        ! Point 24: (200, 700) [rapid], axis_6=0
        CurrentX:=200;
        CurrentY:=700;
        pCurrent.trans:=[-1*CurrentX,CurrentY,SafeZ];
        pCurrent.rot:=OrientZYX(0,20,180);
        pCurrent.robconf:=[1,0,-2,0];
        TcpWorldX:=Bed1Wyong.uframe.trans.x+pCurrent.trans.x;
        CalcTrack:=TcpWorldX;
        IF CurrentY<1000 THEN CalcTrack:=CalcTrack+1500; ENDIF
        IF CurrentY<=1500 THEN
            IF (CalcTrack-TcpWorldX)<MinTrackSep THEN CalcTrack:=TcpWorldX+MinTrackSep; ENDIF
        ENDIF
        IF CalcTrack<TrackMin THEN CalcTrack:=TrackMin; ENDIF
        IF CalcTrack>TrackMax THEN CalcTrack:=TrackMax; ENDIF
        pCurrent.extax:=[CalcTrack,9E+09,9E+09,9E+09,9E+09,9E+09];
        MoveJ pCurrent,v500,z5,tVac\WObj:=Bed1Wyong;

        ! Point 25: (200, 700) [rapid], axis_6=180
        CurrentX:=200;
        CurrentY:=700;
        pCurrent.trans:=[-1*CurrentX,CurrentY,SafeZ];
        pCurrent.rot:=OrientZYX(180,20,180);
        pCurrent.robconf:=[1,0,0,0];
        TcpWorldX:=Bed1Wyong.uframe.trans.x+pCurrent.trans.x;
        CalcTrack:=TcpWorldX;
        IF CurrentY<1000 THEN CalcTrack:=CalcTrack+1500; ENDIF
        IF CurrentY<=1500 THEN
            IF (CalcTrack-TcpWorldX)<MinTrackSep THEN CalcTrack:=TcpWorldX+MinTrackSep; ENDIF
        ENDIF
        IF CalcTrack<TrackMin THEN CalcTrack:=TrackMin; ENDIF
        IF CalcTrack>TrackMax THEN CalcTrack:=TrackMax; ENDIF
        pCurrent.extax:=[CalcTrack,9E+09,9E+09,9E+09,9E+09,9E+09];
        MoveJ pCurrent,v500,z5,tVac\WObj:=Bed1Wyong;

        ! Descend to work height
        pCurrent.trans.z:=WorkZ;
        MoveL pCurrent,v100,z1000,tVac\WObj:=Bed1Wyong;

        ! Point 26: (200, 700) [work], axis_6=180
        CurrentX:=200;
        CurrentY:=700;
        pCurrent.trans:=[-1*CurrentX,CurrentY,WorkZ];
        pCurrent.rot:=OrientZYX(180,20,180);
        pCurrent.robconf:=[1,0,0,0];
        TcpWorldX:=Bed1Wyong.uframe.trans.x+pCurrent.trans.x;
        CalcTrack:=TcpWorldX;
        IF CurrentY<1000 THEN CalcTrack:=CalcTrack+1500; ENDIF
        IF CurrentY<=1500 THEN
            IF (CalcTrack-TcpWorldX)<MinTrackSep THEN CalcTrack:=TcpWorldX+MinTrackSep; ENDIF
        ENDIF
        IF CalcTrack<TrackMin THEN CalcTrack:=TrackMin; ENDIF
        IF CalcTrack>TrackMax THEN CalcTrack:=TrackMax; ENDIF
        pCurrent.extax:=[CalcTrack,9E+09,9E+09,9E+09,9E+09,9E+09];
        MoveL pCurrent,vTravel,z200,tVac\WObj:=Bed1Wyong;

        ! Point 27: (8050, 700) [work], axis_6=180
        CurrentX:=8050;
        CurrentY:=700;
        pCurrent.trans:=[-1*CurrentX,CurrentY,WorkZ];
        pCurrent.rot:=OrientZYX(180,20,180);
        pCurrent.robconf:=[1,0,0,0];
        TcpWorldX:=Bed1Wyong.uframe.trans.x+pCurrent.trans.x;
        CalcTrack:=TcpWorldX;
        IF CurrentY<1000 THEN CalcTrack:=CalcTrack+1500; ENDIF
        IF CurrentY<=1500 THEN
            IF (CalcTrack-TcpWorldX)<MinTrackSep THEN CalcTrack:=TcpWorldX+MinTrackSep; ENDIF
        ENDIF
        IF CalcTrack<TrackMin THEN CalcTrack:=TrackMin; ENDIF
        IF CalcTrack>TrackMax THEN CalcTrack:=TrackMax; ENDIF
        pCurrent.extax:=[CalcTrack,9E+09,9E+09,9E+09,9E+09,9E+09];
        MoveL pCurrent,vTravel,z200,tVac\WObj:=Bed1Wyong;

        ! Point 28: (8050, 500) [rapid], axis_6=180
        CurrentX:=8050;
        CurrentY:=500;
        pCurrent.trans:=[-1*CurrentX,CurrentY,SafeZ];
        pCurrent.rot:=OrientZYX(180,20,180);
        pCurrent.robconf:=[1,0,0,0];
        TcpWorldX:=Bed1Wyong.uframe.trans.x+pCurrent.trans.x;
        CalcTrack:=TcpWorldX;
        IF CurrentY<1000 THEN CalcTrack:=CalcTrack+1500; ENDIF
        IF CurrentY<=1500 THEN
            IF (CalcTrack-TcpWorldX)<MinTrackSep THEN CalcTrack:=TcpWorldX+MinTrackSep; ENDIF
        ENDIF
        IF CalcTrack<TrackMin THEN CalcTrack:=TrackMin; ENDIF
        IF CalcTrack>TrackMax THEN CalcTrack:=TrackMax; ENDIF
        pCurrent.extax:=[CalcTrack,9E+09,9E+09,9E+09,9E+09,9E+09];
        MoveJ pCurrent,v500,z5,tVac\WObj:=Bed1Wyong;

        ! Point 29: (8050, 500) [rapid], axis_6=0
        CurrentX:=8050;
        CurrentY:=500;
        pCurrent.trans:=[-1*CurrentX,CurrentY,SafeZ];
        pCurrent.rot:=OrientZYX(0,20,180);
        pCurrent.robconf:=[1,0,-2,0];
        TcpWorldX:=Bed1Wyong.uframe.trans.x+pCurrent.trans.x;
        CalcTrack:=TcpWorldX;
        IF CurrentY<1000 THEN CalcTrack:=CalcTrack+1500; ENDIF
        IF CurrentY<=1500 THEN
            IF (CalcTrack-TcpWorldX)<MinTrackSep THEN CalcTrack:=TcpWorldX+MinTrackSep; ENDIF
        ENDIF
        IF CalcTrack<TrackMin THEN CalcTrack:=TrackMin; ENDIF
        IF CalcTrack>TrackMax THEN CalcTrack:=TrackMax; ENDIF
        pCurrent.extax:=[CalcTrack,9E+09,9E+09,9E+09,9E+09,9E+09];
        MoveJ pCurrent,v500,z5,tVac\WObj:=Bed1Wyong;

        ! Descend to work height
        pCurrent.trans.z:=WorkZ;
        MoveL pCurrent,v100,z1000,tVac\WObj:=Bed1Wyong;

        ! Point 30: (8050, 500) [work], axis_6=0
        CurrentX:=8050;
        CurrentY:=500;
        pCurrent.trans:=[-1*CurrentX,CurrentY,WorkZ];
        pCurrent.rot:=OrientZYX(0,20,180);
        pCurrent.robconf:=[1,0,-2,0];
        TcpWorldX:=Bed1Wyong.uframe.trans.x+pCurrent.trans.x;
        CalcTrack:=TcpWorldX;
        IF CurrentY<1000 THEN CalcTrack:=CalcTrack+1500; ENDIF
        IF CurrentY<=1500 THEN
            IF (CalcTrack-TcpWorldX)<MinTrackSep THEN CalcTrack:=TcpWorldX+MinTrackSep; ENDIF
        ENDIF
        IF CalcTrack<TrackMin THEN CalcTrack:=TrackMin; ENDIF
        IF CalcTrack>TrackMax THEN CalcTrack:=TrackMax; ENDIF
        pCurrent.extax:=[CalcTrack,9E+09,9E+09,9E+09,9E+09,9E+09];
        MoveL pCurrent,vTravel,z200,tVac\WObj:=Bed1Wyong;

        ! Point 31: (200, 500) [work], axis_6=0
        CurrentX:=200;
        CurrentY:=500;
        pCurrent.trans:=[-1*CurrentX,CurrentY,WorkZ];
        pCurrent.rot:=OrientZYX(0,20,180);
        pCurrent.robconf:=[1,0,-2,0];
        TcpWorldX:=Bed1Wyong.uframe.trans.x+pCurrent.trans.x;
        CalcTrack:=TcpWorldX;
        IF CurrentY<1000 THEN CalcTrack:=CalcTrack+1500; ENDIF
        IF CurrentY<=1500 THEN
            IF (CalcTrack-TcpWorldX)<MinTrackSep THEN CalcTrack:=TcpWorldX+MinTrackSep; ENDIF
        ENDIF
        IF CalcTrack<TrackMin THEN CalcTrack:=TrackMin; ENDIF
        IF CalcTrack>TrackMax THEN CalcTrack:=TrackMax; ENDIF
        pCurrent.extax:=[CalcTrack,9E+09,9E+09,9E+09,9E+09,9E+09];
        MoveL pCurrent,vTravel,z200,tVac\WObj:=Bed1Wyong;

        ! Point 32: (200, 400) [rapid], axis_6=0
        CurrentX:=200;
        CurrentY:=400;
        pCurrent.trans:=[-1*CurrentX,CurrentY,SafeZ];
        pCurrent.rot:=OrientZYX(0,20,180);
        pCurrent.robconf:=[1,0,-2,0];
        TcpWorldX:=Bed1Wyong.uframe.trans.x+pCurrent.trans.x;
        CalcTrack:=TcpWorldX;
        IF CurrentY<1000 THEN CalcTrack:=CalcTrack+1500; ENDIF
        IF CurrentY<=1500 THEN
            IF (CalcTrack-TcpWorldX)<MinTrackSep THEN CalcTrack:=TcpWorldX+MinTrackSep; ENDIF
        ENDIF
        IF CalcTrack<TrackMin THEN CalcTrack:=TrackMin; ENDIF
        IF CalcTrack>TrackMax THEN CalcTrack:=TrackMax; ENDIF
        pCurrent.extax:=[CalcTrack,9E+09,9E+09,9E+09,9E+09,9E+09];
        MoveJ pCurrent,v500,z5,tVac\WObj:=Bed1Wyong;

        ! Point 33: (200, 400) [rapid], axis_6=180
        CurrentX:=200;
        CurrentY:=400;
        pCurrent.trans:=[-1*CurrentX,CurrentY,SafeZ];
        pCurrent.rot:=OrientZYX(180,20,180);
        pCurrent.robconf:=[1,0,0,0];
        TcpWorldX:=Bed1Wyong.uframe.trans.x+pCurrent.trans.x;
        CalcTrack:=TcpWorldX;
        IF CurrentY<1000 THEN CalcTrack:=CalcTrack+1500; ENDIF
        IF CurrentY<=1500 THEN
            IF (CalcTrack-TcpWorldX)<MinTrackSep THEN CalcTrack:=TcpWorldX+MinTrackSep; ENDIF
        ENDIF
        IF CalcTrack<TrackMin THEN CalcTrack:=TrackMin; ENDIF
        IF CalcTrack>TrackMax THEN CalcTrack:=TrackMax; ENDIF
        pCurrent.extax:=[CalcTrack,9E+09,9E+09,9E+09,9E+09,9E+09];
        MoveJ pCurrent,v500,z5,tVac\WObj:=Bed1Wyong;

        ! Descend to work height
        pCurrent.trans.z:=WorkZ;
        MoveL pCurrent,v100,z1000,tVac\WObj:=Bed1Wyong;

        ! Point 34: (200, 400) [work], axis_6=180
        CurrentX:=200;
        CurrentY:=400;
        pCurrent.trans:=[-1*CurrentX,CurrentY,WorkZ];
        pCurrent.rot:=OrientZYX(180,20,180);
        pCurrent.robconf:=[1,0,0,0];
        TcpWorldX:=Bed1Wyong.uframe.trans.x+pCurrent.trans.x;
        CalcTrack:=TcpWorldX;
        IF CurrentY<1000 THEN CalcTrack:=CalcTrack+1500; ENDIF
        IF CurrentY<=1500 THEN
            IF (CalcTrack-TcpWorldX)<MinTrackSep THEN CalcTrack:=TcpWorldX+MinTrackSep; ENDIF
        ENDIF
        IF CalcTrack<TrackMin THEN CalcTrack:=TrackMin; ENDIF
        IF CalcTrack>TrackMax THEN CalcTrack:=TrackMax; ENDIF
        pCurrent.extax:=[CalcTrack,9E+09,9E+09,9E+09,9E+09,9E+09];
        MoveL pCurrent,vTravel,z200,tVac\WObj:=Bed1Wyong;

        ! Point 35: (8050, 400) [work], axis_6=180
        CurrentX:=8050;
        CurrentY:=400;
        pCurrent.trans:=[-1*CurrentX,CurrentY,WorkZ];
        pCurrent.rot:=OrientZYX(180,20,180);
        pCurrent.robconf:=[1,0,0,0];
        TcpWorldX:=Bed1Wyong.uframe.trans.x+pCurrent.trans.x;
        CalcTrack:=TcpWorldX;
        IF CurrentY<1000 THEN CalcTrack:=CalcTrack+1500; ENDIF
        IF CurrentY<=1500 THEN
            IF (CalcTrack-TcpWorldX)<MinTrackSep THEN CalcTrack:=TcpWorldX+MinTrackSep; ENDIF
        ENDIF
        IF CalcTrack<TrackMin THEN CalcTrack:=TrackMin; ENDIF
        IF CalcTrack>TrackMax THEN CalcTrack:=TrackMax; ENDIF
        pCurrent.extax:=[CalcTrack,9E+09,9E+09,9E+09,9E+09,9E+09];
        MoveL pCurrent,vTravel,z200,tVac\WObj:=Bed1Wyong;


        ! Lift to safe height (before motor off for smooth blend)
        pCurrent.trans.z:=WorkZ+500;
        MoveL pCurrent,v200,z1000,tVac\WObj:=Bed1Wyong;
        Vac_off;

        ! Return tool and go home
        TPWrite "Py2Vac: Dropping off tool...";
        Vac_Dropoff;
        Home FALSE;

        TPWrite "========================================";
        TPWrite "Py2Vac: COMPLETE";
        TPWrite "========================================";

    ERROR
        Vac_off;
        TPWrite "Py2Vac ERROR: " \Num:=ERRNO;
        RAISE;
    ENDPROC

    PROC Py2Pan()
        ! Py2Pan - Generated by Onyx Tool Class
        ! Workzone: panel
        ! Area: (500,500) to (1900,1800)
        ! Z = 451mm
        ! Step: 300mm

        VAR robtarget pCurrent;
        VAR jointtarget CurrentJoints;
        VAR robtarget CurrentPos;
        VAR num WorkZ:=451;
        VAR num SafeZ:=651;
        VAR num CurrentX:=0;
        VAR num CurrentY:=0;
        VAR speeddata vTravel:=[100,500,5000,1000];
        VAR num TrackMin:=-300;
        VAR num TrackMax:=10050;
        VAR num CalcTrack:=0;
        VAR zonedata z1000:=[FALSE,1000,1500,1500,150,1500,150];
        VAR num PanForce:=0;
        VAR bool bFCActive:=FALSE;

        TPWrite "========================================";
        TPWrite "Py2Pan: Starting";
        TPWrite "========================================";
        TPWrite "Workzone: panel";
        TPWrite "WorkZ=" \Num:=WorkZ;

        ! Get helicopter tool (Pan attaches to it)
        UpdateToolNum;
        IF ToolNum<>2 THEN
            TPWrite "Py2Pan: Getting helicopter...";
            Home TRUE;
            Heli_Pickup;
        ELSE
            CurrentJoints:=CJointT();
            CurrentPos:=CalcRobT(CurrentJoints,tHeli\WObj:=wobj0);
            IF (CurrentPos.trans.x)>8000 AND CurrentPos.trans.z<400 THEN
                MoveL Offs(CurrentPos,0,0,(400-CurrentPos.trans.z)),v100,z5,tHeli;
            ENDIF
        ENDIF

        ! Set blade angle = 0 for pan
        HeliBlade_Angle 0;

        ! Start blade rotation
        TPWrite "Py2Pan: Starting blades at " \Num:=80;
        HeliBladeSpeed 80,"REV";
        TPWrite "Py2Pan: Blades motor on";
        WaitTime 5;

        ! ========================================
        ! Pattern Execution: 24 points
        ! ========================================

        ! Point 1: (500, 1800) [rapid]
        CurrentX:=500;
        CurrentY:=1800;
        pCurrent.trans:=[-1*CurrentX,CurrentY,SafeZ];
        pCurrent.rot:=OrientZYX(0,0,180);
        pCurrent.robconf:=[1,0,-2,0];
        CalcTrack:=Bed1Wyong.uframe.trans.x+pCurrent.trans.x;
        IF CurrentY<1000 THEN CalcTrack:=CalcTrack+1200; ENDIF
        IF CalcTrack<TrackMin THEN CalcTrack:=TrackMin; ENDIF
        IF CalcTrack>TrackMax THEN CalcTrack:=TrackMax; ENDIF
        pCurrent.extax:=[CalcTrack,9E+09,9E+09,9E+09,9E+09,9E+09];
        MoveJ pCurrent,v500,z5,tHeli\WObj:=Bed1Wyong;

        ! Descend to work height
        pCurrent.trans.z:=WorkZ;
        MoveL pCurrent,v100,z1000,tHeli\WObj:=Bed1Wyong;

        ! Point 2: (1900, 1800) [work]
        CurrentX:=1900;
        CurrentY:=1800;
        pCurrent.trans:=[-1*CurrentX,CurrentY,WorkZ];
        pCurrent.rot:=OrientZYX(0,0,180);
        pCurrent.robconf:=[1,0,-2,0];
        CalcTrack:=Bed1Wyong.uframe.trans.x+pCurrent.trans.x;
        IF CurrentY<1000 THEN CalcTrack:=CalcTrack+1200; ENDIF
        IF CalcTrack<TrackMin THEN CalcTrack:=TrackMin; ENDIF
        IF CalcTrack>TrackMax THEN CalcTrack:=TrackMax; ENDIF
        pCurrent.extax:=[CalcTrack,9E+09,9E+09,9E+09,9E+09,9E+09];
        MoveL pCurrent,vTravel,z200,tHeli\WObj:=Bed1Wyong;

        ! Point 3: (1900, 1500) [work]
        CurrentX:=1900;
        CurrentY:=1500;
        pCurrent.trans:=[-1*CurrentX,CurrentY,WorkZ];
        pCurrent.rot:=OrientZYX(0,0,180);
        pCurrent.robconf:=[1,0,-2,0];
        CalcTrack:=Bed1Wyong.uframe.trans.x+pCurrent.trans.x;
        IF CurrentY<1000 THEN CalcTrack:=CalcTrack+1200; ENDIF
        IF CalcTrack<TrackMin THEN CalcTrack:=TrackMin; ENDIF
        IF CalcTrack>TrackMax THEN CalcTrack:=TrackMax; ENDIF
        pCurrent.extax:=[CalcTrack,9E+09,9E+09,9E+09,9E+09,9E+09];
        MoveL pCurrent,vTravel,z200,tHeli\WObj:=Bed1Wyong;

        ! Point 4: (500, 1500) [work]
        CurrentX:=500;
        CurrentY:=1500;
        pCurrent.trans:=[-1*CurrentX,CurrentY,WorkZ];
        pCurrent.rot:=OrientZYX(0,0,180);
        pCurrent.robconf:=[1,0,-2,0];
        CalcTrack:=Bed1Wyong.uframe.trans.x+pCurrent.trans.x;
        IF CurrentY<1000 THEN CalcTrack:=CalcTrack+1200; ENDIF
        IF CalcTrack<TrackMin THEN CalcTrack:=TrackMin; ENDIF
        IF CalcTrack>TrackMax THEN CalcTrack:=TrackMax; ENDIF
        pCurrent.extax:=[CalcTrack,9E+09,9E+09,9E+09,9E+09,9E+09];
        MoveL pCurrent,vTravel,z200,tHeli\WObj:=Bed1Wyong;

        ! Point 5: (500, 1200) [work]
        CurrentX:=500;
        CurrentY:=1200;
        pCurrent.trans:=[-1*CurrentX,CurrentY,WorkZ];
        pCurrent.rot:=OrientZYX(0,0,180);
        pCurrent.robconf:=[1,0,-2,0];
        CalcTrack:=Bed1Wyong.uframe.trans.x+pCurrent.trans.x;
        IF CurrentY<1000 THEN CalcTrack:=CalcTrack+1200; ENDIF
        IF CalcTrack<TrackMin THEN CalcTrack:=TrackMin; ENDIF
        IF CalcTrack>TrackMax THEN CalcTrack:=TrackMax; ENDIF
        pCurrent.extax:=[CalcTrack,9E+09,9E+09,9E+09,9E+09,9E+09];
        MoveL pCurrent,vTravel,z200,tHeli\WObj:=Bed1Wyong;

        ! Point 6: (1900, 1200) [work]
        CurrentX:=1900;
        CurrentY:=1200;
        pCurrent.trans:=[-1*CurrentX,CurrentY,WorkZ];
        pCurrent.rot:=OrientZYX(0,0,180);
        pCurrent.robconf:=[1,0,-2,0];
        CalcTrack:=Bed1Wyong.uframe.trans.x+pCurrent.trans.x;
        IF CurrentY<1000 THEN CalcTrack:=CalcTrack+1200; ENDIF
        IF CalcTrack<TrackMin THEN CalcTrack:=TrackMin; ENDIF
        IF CalcTrack>TrackMax THEN CalcTrack:=TrackMax; ENDIF
        pCurrent.extax:=[CalcTrack,9E+09,9E+09,9E+09,9E+09,9E+09];
        MoveL pCurrent,vTravel,z200,tHeli\WObj:=Bed1Wyong;

        ! Point 7: (1900, 900) [work]
        CurrentX:=1900;
        CurrentY:=900;
        pCurrent.trans:=[-1*CurrentX,CurrentY,WorkZ];
        pCurrent.rot:=OrientZYX(0,0,180);
        pCurrent.robconf:=[1,0,-2,0];
        CalcTrack:=Bed1Wyong.uframe.trans.x+pCurrent.trans.x;
        IF CurrentY<1000 THEN CalcTrack:=CalcTrack+1200; ENDIF
        IF CalcTrack<TrackMin THEN CalcTrack:=TrackMin; ENDIF
        IF CalcTrack>TrackMax THEN CalcTrack:=TrackMax; ENDIF
        pCurrent.extax:=[CalcTrack,9E+09,9E+09,9E+09,9E+09,9E+09];
        MoveL pCurrent,vTravel,z200,tHeli\WObj:=Bed1Wyong;

        ! Point 8: (500, 900) [work]
        CurrentX:=500;
        CurrentY:=900;
        pCurrent.trans:=[-1*CurrentX,CurrentY,WorkZ];
        pCurrent.rot:=OrientZYX(0,0,180);
        pCurrent.robconf:=[1,0,-2,0];
        CalcTrack:=Bed1Wyong.uframe.trans.x+pCurrent.trans.x;
        IF CurrentY<1000 THEN CalcTrack:=CalcTrack+1200; ENDIF
        IF CalcTrack<TrackMin THEN CalcTrack:=TrackMin; ENDIF
        IF CalcTrack>TrackMax THEN CalcTrack:=TrackMax; ENDIF
        pCurrent.extax:=[CalcTrack,9E+09,9E+09,9E+09,9E+09,9E+09];
        MoveL pCurrent,vTravel,z200,tHeli\WObj:=Bed1Wyong;

        ! Point 9: (500, 600) [work]
        CurrentX:=500;
        CurrentY:=600;
        pCurrent.trans:=[-1*CurrentX,CurrentY,WorkZ];
        pCurrent.rot:=OrientZYX(0,0,180);
        pCurrent.robconf:=[1,0,-2,0];
        CalcTrack:=Bed1Wyong.uframe.trans.x+pCurrent.trans.x;
        IF CurrentY<1000 THEN CalcTrack:=CalcTrack+1200; ENDIF
        IF CalcTrack<TrackMin THEN CalcTrack:=TrackMin; ENDIF
        IF CalcTrack>TrackMax THEN CalcTrack:=TrackMax; ENDIF
        pCurrent.extax:=[CalcTrack,9E+09,9E+09,9E+09,9E+09,9E+09];
        MoveL pCurrent,vTravel,z200,tHeli\WObj:=Bed1Wyong;

        ! Point 10: (1900, 600) [work]
        CurrentX:=1900;
        CurrentY:=600;
        pCurrent.trans:=[-1*CurrentX,CurrentY,WorkZ];
        pCurrent.rot:=OrientZYX(0,0,180);
        pCurrent.robconf:=[1,0,-2,0];
        CalcTrack:=Bed1Wyong.uframe.trans.x+pCurrent.trans.x;
        IF CurrentY<1000 THEN CalcTrack:=CalcTrack+1200; ENDIF
        IF CalcTrack<TrackMin THEN CalcTrack:=TrackMin; ENDIF
        IF CalcTrack>TrackMax THEN CalcTrack:=TrackMax; ENDIF
        pCurrent.extax:=[CalcTrack,9E+09,9E+09,9E+09,9E+09,9E+09];
        MoveL pCurrent,vTravel,z200,tHeli\WObj:=Bed1Wyong;

        ! Point 11: (1900, 500) [work]
        CurrentX:=1900;
        CurrentY:=500;
        pCurrent.trans:=[-1*CurrentX,CurrentY,WorkZ];
        pCurrent.rot:=OrientZYX(0,0,180);
        pCurrent.robconf:=[1,0,-2,0];
        CalcTrack:=Bed1Wyong.uframe.trans.x+pCurrent.trans.x;
        IF CurrentY<1000 THEN CalcTrack:=CalcTrack+1200; ENDIF
        IF CalcTrack<TrackMin THEN CalcTrack:=TrackMin; ENDIF
        IF CalcTrack>TrackMax THEN CalcTrack:=TrackMax; ENDIF
        pCurrent.extax:=[CalcTrack,9E+09,9E+09,9E+09,9E+09,9E+09];
        MoveL pCurrent,vTravel,z200,tHeli\WObj:=Bed1Wyong;

        ! Point 12: (500, 500) [work]
        CurrentX:=500;
        CurrentY:=500;
        pCurrent.trans:=[-1*CurrentX,CurrentY,WorkZ];
        pCurrent.rot:=OrientZYX(0,0,180);
        pCurrent.robconf:=[1,0,-2,0];
        CalcTrack:=Bed1Wyong.uframe.trans.x+pCurrent.trans.x;
        IF CurrentY<1000 THEN CalcTrack:=CalcTrack+1200; ENDIF
        IF CalcTrack<TrackMin THEN CalcTrack:=TrackMin; ENDIF
        IF CalcTrack>TrackMax THEN CalcTrack:=TrackMax; ENDIF
        pCurrent.extax:=[CalcTrack,9E+09,9E+09,9E+09,9E+09,9E+09];
        MoveL pCurrent,vTravel,z200,tHeli\WObj:=Bed1Wyong;

        ! Point 13: (500, 500) [work]
        CurrentX:=500;
        CurrentY:=500;
        pCurrent.trans:=[-1*CurrentX,CurrentY,WorkZ];
        pCurrent.rot:=OrientZYX(0,0,180);
        pCurrent.robconf:=[1,0,-2,0];
        CalcTrack:=Bed1Wyong.uframe.trans.x+pCurrent.trans.x;
        IF CurrentY<1000 THEN CalcTrack:=CalcTrack+1200; ENDIF
        IF CalcTrack<TrackMin THEN CalcTrack:=TrackMin; ENDIF
        IF CalcTrack>TrackMax THEN CalcTrack:=TrackMax; ENDIF
        pCurrent.extax:=[CalcTrack,9E+09,9E+09,9E+09,9E+09,9E+09];
        MoveL pCurrent,vTravel,z200,tHeli\WObj:=Bed1Wyong;

        ! Point 14: (500, 1800) [work]
        CurrentX:=500;
        CurrentY:=1800;
        pCurrent.trans:=[-1*CurrentX,CurrentY,WorkZ];
        pCurrent.rot:=OrientZYX(0,0,180);
        pCurrent.robconf:=[1,0,-2,0];
        CalcTrack:=Bed1Wyong.uframe.trans.x+pCurrent.trans.x;
        IF CurrentY<1000 THEN CalcTrack:=CalcTrack+1200; ENDIF
        IF CalcTrack<TrackMin THEN CalcTrack:=TrackMin; ENDIF
        IF CalcTrack>TrackMax THEN CalcTrack:=TrackMax; ENDIF
        pCurrent.extax:=[CalcTrack,9E+09,9E+09,9E+09,9E+09,9E+09];
        MoveL pCurrent,vTravel,z200,tHeli\WObj:=Bed1Wyong;

        ! Point 15: (800, 1800) [work]
        CurrentX:=800;
        CurrentY:=1800;
        pCurrent.trans:=[-1*CurrentX,CurrentY,WorkZ];
        pCurrent.rot:=OrientZYX(0,0,180);
        pCurrent.robconf:=[1,0,-2,0];
        CalcTrack:=Bed1Wyong.uframe.trans.x+pCurrent.trans.x;
        IF CurrentY<1000 THEN CalcTrack:=CalcTrack+1200; ENDIF
        IF CalcTrack<TrackMin THEN CalcTrack:=TrackMin; ENDIF
        IF CalcTrack>TrackMax THEN CalcTrack:=TrackMax; ENDIF
        pCurrent.extax:=[CalcTrack,9E+09,9E+09,9E+09,9E+09,9E+09];
        MoveL pCurrent,vTravel,z200,tHeli\WObj:=Bed1Wyong;

        ! Point 16: (800, 500) [work]
        CurrentX:=800;
        CurrentY:=500;
        pCurrent.trans:=[-1*CurrentX,CurrentY,WorkZ];
        pCurrent.rot:=OrientZYX(0,0,180);
        pCurrent.robconf:=[1,0,-2,0];
        CalcTrack:=Bed1Wyong.uframe.trans.x+pCurrent.trans.x;
        IF CurrentY<1000 THEN CalcTrack:=CalcTrack+1200; ENDIF
        IF CalcTrack<TrackMin THEN CalcTrack:=TrackMin; ENDIF
        IF CalcTrack>TrackMax THEN CalcTrack:=TrackMax; ENDIF
        pCurrent.extax:=[CalcTrack,9E+09,9E+09,9E+09,9E+09,9E+09];
        MoveL pCurrent,vTravel,z200,tHeli\WObj:=Bed1Wyong;

        ! Point 17: (1100, 500) [work]
        CurrentX:=1100;
        CurrentY:=500;
        pCurrent.trans:=[-1*CurrentX,CurrentY,WorkZ];
        pCurrent.rot:=OrientZYX(0,0,180);
        pCurrent.robconf:=[1,0,-2,0];
        CalcTrack:=Bed1Wyong.uframe.trans.x+pCurrent.trans.x;
        IF CurrentY<1000 THEN CalcTrack:=CalcTrack+1200; ENDIF
        IF CalcTrack<TrackMin THEN CalcTrack:=TrackMin; ENDIF
        IF CalcTrack>TrackMax THEN CalcTrack:=TrackMax; ENDIF
        pCurrent.extax:=[CalcTrack,9E+09,9E+09,9E+09,9E+09,9E+09];
        MoveL pCurrent,vTravel,z200,tHeli\WObj:=Bed1Wyong;

        ! Point 18: (1100, 1800) [work]
        CurrentX:=1100;
        CurrentY:=1800;
        pCurrent.trans:=[-1*CurrentX,CurrentY,WorkZ];
        pCurrent.rot:=OrientZYX(0,0,180);
        pCurrent.robconf:=[1,0,-2,0];
        CalcTrack:=Bed1Wyong.uframe.trans.x+pCurrent.trans.x;
        IF CurrentY<1000 THEN CalcTrack:=CalcTrack+1200; ENDIF
        IF CalcTrack<TrackMin THEN CalcTrack:=TrackMin; ENDIF
        IF CalcTrack>TrackMax THEN CalcTrack:=TrackMax; ENDIF
        pCurrent.extax:=[CalcTrack,9E+09,9E+09,9E+09,9E+09,9E+09];
        MoveL pCurrent,vTravel,z200,tHeli\WObj:=Bed1Wyong;

        ! Point 19: (1400, 1800) [work]
        CurrentX:=1400;
        CurrentY:=1800;
        pCurrent.trans:=[-1*CurrentX,CurrentY,WorkZ];
        pCurrent.rot:=OrientZYX(0,0,180);
        pCurrent.robconf:=[1,0,-2,0];
        CalcTrack:=Bed1Wyong.uframe.trans.x+pCurrent.trans.x;
        IF CurrentY<1000 THEN CalcTrack:=CalcTrack+1200; ENDIF
        IF CalcTrack<TrackMin THEN CalcTrack:=TrackMin; ENDIF
        IF CalcTrack>TrackMax THEN CalcTrack:=TrackMax; ENDIF
        pCurrent.extax:=[CalcTrack,9E+09,9E+09,9E+09,9E+09,9E+09];
        MoveL pCurrent,vTravel,z200,tHeli\WObj:=Bed1Wyong;

        ! Point 20: (1400, 500) [work]
        CurrentX:=1400;
        CurrentY:=500;
        pCurrent.trans:=[-1*CurrentX,CurrentY,WorkZ];
        pCurrent.rot:=OrientZYX(0,0,180);
        pCurrent.robconf:=[1,0,-2,0];
        CalcTrack:=Bed1Wyong.uframe.trans.x+pCurrent.trans.x;
        IF CurrentY<1000 THEN CalcTrack:=CalcTrack+1200; ENDIF
        IF CalcTrack<TrackMin THEN CalcTrack:=TrackMin; ENDIF
        IF CalcTrack>TrackMax THEN CalcTrack:=TrackMax; ENDIF
        pCurrent.extax:=[CalcTrack,9E+09,9E+09,9E+09,9E+09,9E+09];
        MoveL pCurrent,vTravel,z200,tHeli\WObj:=Bed1Wyong;

        ! Point 21: (1700, 500) [work]
        CurrentX:=1700;
        CurrentY:=500;
        pCurrent.trans:=[-1*CurrentX,CurrentY,WorkZ];
        pCurrent.rot:=OrientZYX(0,0,180);
        pCurrent.robconf:=[1,0,-2,0];
        CalcTrack:=Bed1Wyong.uframe.trans.x+pCurrent.trans.x;
        IF CurrentY<1000 THEN CalcTrack:=CalcTrack+1200; ENDIF
        IF CalcTrack<TrackMin THEN CalcTrack:=TrackMin; ENDIF
        IF CalcTrack>TrackMax THEN CalcTrack:=TrackMax; ENDIF
        pCurrent.extax:=[CalcTrack,9E+09,9E+09,9E+09,9E+09,9E+09];
        MoveL pCurrent,vTravel,z200,tHeli\WObj:=Bed1Wyong;

        ! Point 22: (1700, 1800) [work]
        CurrentX:=1700;
        CurrentY:=1800;
        pCurrent.trans:=[-1*CurrentX,CurrentY,WorkZ];
        pCurrent.rot:=OrientZYX(0,0,180);
        pCurrent.robconf:=[1,0,-2,0];
        CalcTrack:=Bed1Wyong.uframe.trans.x+pCurrent.trans.x;
        IF CurrentY<1000 THEN CalcTrack:=CalcTrack+1200; ENDIF
        IF CalcTrack<TrackMin THEN CalcTrack:=TrackMin; ENDIF
        IF CalcTrack>TrackMax THEN CalcTrack:=TrackMax; ENDIF
        pCurrent.extax:=[CalcTrack,9E+09,9E+09,9E+09,9E+09,9E+09];
        MoveL pCurrent,vTravel,z200,tHeli\WObj:=Bed1Wyong;

        ! Point 23: (1900, 1800) [work]
        CurrentX:=1900;
        CurrentY:=1800;
        pCurrent.trans:=[-1*CurrentX,CurrentY,WorkZ];
        pCurrent.rot:=OrientZYX(0,0,180);
        pCurrent.robconf:=[1,0,-2,0];
        CalcTrack:=Bed1Wyong.uframe.trans.x+pCurrent.trans.x;
        IF CurrentY<1000 THEN CalcTrack:=CalcTrack+1200; ENDIF
        IF CalcTrack<TrackMin THEN CalcTrack:=TrackMin; ENDIF
        IF CalcTrack>TrackMax THEN CalcTrack:=TrackMax; ENDIF
        pCurrent.extax:=[CalcTrack,9E+09,9E+09,9E+09,9E+09,9E+09];
        MoveL pCurrent,vTravel,z200,tHeli\WObj:=Bed1Wyong;

        ! Point 24: (1900, 500) [work]
        CurrentX:=1900;
        CurrentY:=500;
        pCurrent.trans:=[-1*CurrentX,CurrentY,WorkZ];
        pCurrent.rot:=OrientZYX(0,0,180);
        pCurrent.robconf:=[1,0,-2,0];
        CalcTrack:=Bed1Wyong.uframe.trans.x+pCurrent.trans.x;
        IF CurrentY<1000 THEN CalcTrack:=CalcTrack+1200; ENDIF
        IF CalcTrack<TrackMin THEN CalcTrack:=TrackMin; ENDIF
        IF CalcTrack>TrackMax THEN CalcTrack:=TrackMax; ENDIF
        pCurrent.extax:=[CalcTrack,9E+09,9E+09,9E+09,9E+09,9E+09];
        MoveL pCurrent,vTravel,z200,tHeli\WObj:=Bed1Wyong;


        ! Lift to safe height (before motor off for smooth blend)
        pCurrent.trans.z:=WorkZ+500;
        MoveL pCurrent,v200,z1000,tHeli\WObj:=Bed1Wyong;
        ! Stop blade rotation
        HeliBladeSpeed 0,"REV";
        WaitTime 1;

        ! Return tool and go home
        TPWrite "Py2Pan: Dropping off helicopter...";
        Heli_Dropoff;
        Home FALSE;

        TPWrite "========================================";
        TPWrite "Py2Pan: COMPLETE";
        TPWrite "========================================";

    ERROR
        HeliBladeSpeed 0,"REV";
        IF bFCActive THEN
            FCPressEnd Offs(CurrentPos,0,0,100),v50,\DeactOnly,tHeli\WObj:=Bed1Wyong;
        ENDIF
        RAISE;
    ENDPROC

    PROC Py2VS()
        ! Py2VS - Generated by Onyx Tool Class
        ! Workzone: panel
        ! Area: (550,550) to (1850,1750)
        ! Z = 450mm
        ! Step: 200mm

        VAR robtarget pCurrent;
        VAR jointtarget CurrentJoints;
        VAR robtarget CurrentPos;
        VAR num WorkZ:=450;
        VAR num SafeZ:=650;
        VAR num CurrentX:=0;
        VAR num CurrentY:=0;
        VAR speeddata vTravel:=[75,15,2000,15];
        VAR num TrackMin:=-300;
        VAR num TrackMax:=10050;
        VAR num CalcTrack:=0;
        VAR zonedata z1000:=[FALSE,1000,1500,1500,150,1500,150];

        TPWrite "========================================";
        TPWrite "Py2VS: Starting";
        TPWrite "========================================";
        TPWrite "Workzone: panel";
        TPWrite "WorkZ=" \Num:=WorkZ;

        ! Get tool if needed
        UpdateToolNum;
        IF ToolNum<>3 THEN
            TPWrite "Py2VS: Getting tool...";
            Home TRUE;
            VS_Pickup;
        ELSE
            CurrentJoints:=CJointT();
            CurrentPos:=CalcRobT(CurrentJoints,tVS\WObj:=wobj0);
            IF (CurrentPos.trans.x)>8000 AND CurrentPos.trans.z<400 THEN
                MoveL Offs(CurrentPos,0,0,(400-CurrentPos.trans.z)),v100,z5,tVS;
            ENDIF
        ENDIF

        ! ========================================
        ! Pattern Execution: 4 points
        ! Force Monitoring: DISABLED
        ! ========================================

        ! Use VS tool's orientation from pickup end position (pVSHome3)
        ! This prevents 180 degree rotation when moving to work surface
        pCurrent.rot:=pVSHome3.rot;

        ! Point 1: (140, 2100) [rapid]
        CurrentX:=140;
        CurrentY:=2100;
        pCurrent.trans:=[-1*CurrentX,CurrentY,SafeZ];
        pCurrent.robconf:=[1,0,1,0];
        CalcTrack:=Bed1Wyong.uframe.trans.x+pCurrent.trans.x;
        IF CurrentY<1000 THEN CalcTrack:=CalcTrack+1200; ENDIF
        IF CalcTrack<TrackMin THEN CalcTrack:=TrackMin; ENDIF
        IF CalcTrack>TrackMax THEN CalcTrack:=TrackMax; ENDIF
        pCurrent.extax:=[CalcTrack,9E+09,9E+09,9E+09,9E+09,9E+09];
        MoveJ pCurrent,v500,z5,tVS\WObj:=Bed1Wyong;

        ! Turn on vibrating screed after positioning
        TPWrite "Py2VS: Starting screed...";
        VS_on;

        ! Point 2: (190, 2100) [work]
        CurrentX:=190;
        CurrentY:=2100;
        pCurrent.trans:=[-1*CurrentX,CurrentY,WorkZ];
        pCurrent.robconf:=[1,0,1,0];
        CalcTrack:=Bed1Wyong.uframe.trans.x+pCurrent.trans.x;
        IF CurrentY<1000 THEN CalcTrack:=CalcTrack+1200; ENDIF
        IF CalcTrack<TrackMin THEN CalcTrack:=TrackMin; ENDIF
        IF CalcTrack>TrackMax THEN CalcTrack:=TrackMax; ENDIF
        pCurrent.extax:=[CalcTrack,9E+09,9E+09,9E+09,9E+09,9E+09];
        MoveL pCurrent,vTravel,z200,tVS\WObj:=Bed1Wyong;

        ! Point 3: (2210, 2100) [work]
        CurrentX:=2210;
        CurrentY:=2100;
        pCurrent.trans:=[-1*CurrentX,CurrentY,WorkZ];
        pCurrent.robconf:=[1,0,1,0];
        CalcTrack:=Bed1Wyong.uframe.trans.x+pCurrent.trans.x;
        IF CurrentY<1000 THEN CalcTrack:=CalcTrack+1200; ENDIF
        IF CalcTrack<TrackMin THEN CalcTrack:=TrackMin; ENDIF
        IF CalcTrack>TrackMax THEN CalcTrack:=TrackMax; ENDIF
        pCurrent.extax:=[CalcTrack,9E+09,9E+09,9E+09,9E+09,9E+09];
        MoveL pCurrent,vTravel,z200,tVS\WObj:=Bed1Wyong;

        ! Point 4: (2260, 2100) [rapid]
        CurrentX:=2260;
        CurrentY:=2100;
        pCurrent.trans:=[-1*CurrentX,CurrentY,SafeZ];
        pCurrent.robconf:=[1,0,1,0];
        CalcTrack:=Bed1Wyong.uframe.trans.x+pCurrent.trans.x;
        IF CurrentY<1000 THEN CalcTrack:=CalcTrack+1200; ENDIF
        IF CalcTrack<TrackMin THEN CalcTrack:=TrackMin; ENDIF
        IF CalcTrack>TrackMax THEN CalcTrack:=TrackMax; ENDIF
        pCurrent.extax:=[CalcTrack,9E+09,9E+09,9E+09,9E+09,9E+09];
        MoveJ pCurrent,v500,z5,tVS\WObj:=Bed1Wyong;


        ! Lift to safe height (before motor off for smooth blend)
        pCurrent.trans.z:=WorkZ+500;
        MoveL pCurrent,v200,z1000,tVS\WObj:=Bed1Wyong;
        VS_off;

        ! Return tool and go home
        TPWrite "Py2VS: Dropping off tool...";
        VS_Dropoff;
        Home FALSE;

        TPWrite "========================================";
        TPWrite "Py2VS: COMPLETE";
        TPWrite "========================================";

    ERROR
        VS_off;
        TPWrite "Py2VS ERROR: " \Num:=ERRNO;
        RAISE;
    ENDPROC


    PROC SeqBedClean()
        ! SeqBedClean - Bed Cleaning Sequence
        ! Runs: Vacuum -> Polish
        ! Generated by Onyx Toolpath Generator v2

        TPWrite "========================================";
        TPWrite "SeqBedClean: Starting Bed Clean Sequence";
        TPWrite "========================================";
        TPWrite "Step 1: Vacuum";
        TPWrite "Step 2: Polish";
        TPWrite "========================================";

        ! Step 1: Vacuum the bed
        TPWrite "SeqBedClean: Starting vacuum...";
        Py2Vac;
        TPWrite "SeqBedClean: Vacuum complete";

        ! Step 2: Polish the bed
        TPWrite "SeqBedClean: Starting polish...";
        Py2Polish;
        TPWrite "SeqBedClean: Polish complete";

        TPWrite "========================================";
        TPWrite "SeqBedClean: SEQUENCE COMPLETE";
        TPWrite "========================================";

    ERROR
        TPWrite "SeqBedClean ERROR: " \Num:=ERRNO;
        RAISE;
    ENDPROC


    ! ========== END PY2 GENERATED PROCEDURES ==========

ENDMODULE
